FUNCTION_BLOCK ABSTRACT FB_CommandChange EXTENDS FB_BaseComponent IMPLEMENTS ITF_CommandChange
VAR
	itfSaMController				: ITF_SaMControllerCommandChange;
	
END_VAR

(*			
	EVERDE sp. z o.o.
	Rafał Osajda		03.11.2025		TC 4024.66
	Test czy można zmienić stan lub tryb i zwraca czy można i uruchamia zmianę
*)
METHOD PUBLIC Execute : BOOL
VAR_INPUT
END_VAR
IF (TRUE) THEN
	THIS^.itfSaMController.ChangeStateTo (eNewState := E_SaMStates.Aborting);
END_IF
END_METHOD

(*			
	EVERDE sp. z o.o.
	Rafał Osajda		03.11.2025		TC 4024.66
	Podłączenie sterowania do SaMController
*)
METHOD PUBLIC LinkSaMCotroller : BOOL
VAR_INPUT
	itfSaMController		: ITF_SaMControllerCommandChange;
END_VAR
THIS^.itfSaMController		:= itfSaMController;
END_METHOD

END_FUNCTION_BLOCK

(* stored: Version 1.1.0.1
   POU FB_CommandChange: Id {2908caa6-01fe-00f1-181a-1acec604552c}, SpecialFunc None
   Method Execute: Id {3e1ea8aa-acdf-0fb7-0ce9-e01f53a6e468}
   Method LinkSaMCotroller: Id {a1ee9fff-ed2f-0895-2d8b-6d4b59c9eb07} *)
